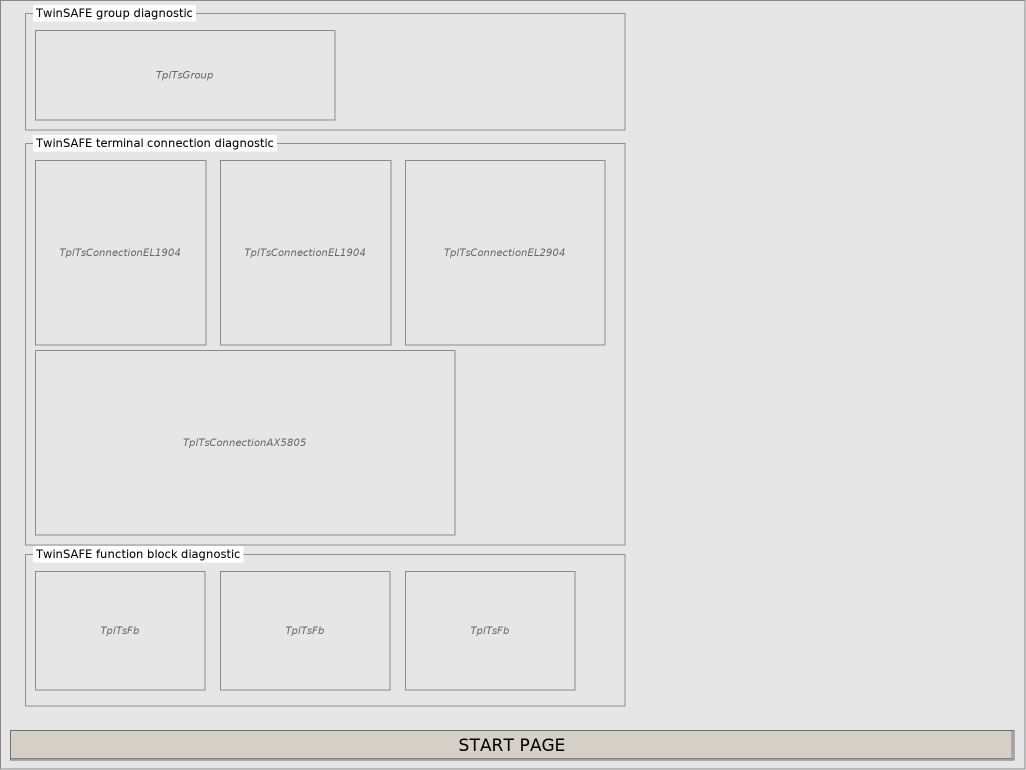
VISUALIZATION HmiTwinSAFEDiagnostic  // 1026x770
    Rectangle (0,0 1024x768)
    GroupBox (25,5 600x125), "TwinSAFE group diagnostic"
        Frame (10,25 300x90)
            shows TplTsGroup(stGroupDiag := TwinSAFE.fbSafeGroup1)
    GroupBox (25,135 600x410), "TwinSAFE terminal connection diagnostic"
        Frame (195,25 171x185)
            shows TplTsConnectionEL1904(stConnectionDiag := TwinSAFE.fbSafeConnectionEL1904_2_Group1)
        Frame (380,25 200x185)
            shows TplTsConnectionEL2904(stConnectionDiag := TwinSAFE.fbSafeConnectionEL2904_1_Group1)
        Frame (10,25 171x185)
            shows TplTsConnectionEL1904(stConnectionDiag := TwinSAFE.fbSafeConnectionEL1904_1_Group1)
        Frame (10,215 420x185)
            shows TplTsConnectionAX5805(stConnectionDiag := TwinSAFE.fbSafeConnectionAX5805_1_Group1)
    GroupBox (25,546 600x160), "TwinSAFE function block diagnostic"
        Frame (10,25 170x119)
            shows TplTsFb(stfbDiag := TwinSAFE.fbSafeFB_1_Group1)
        Frame (195,25 170x119)
            shows TplTsFb(stfbDiag := TwinSAFE.fbSafeFB_2_Group1)
        Frame (380,25 170x119)
            shows TplTsFb(stfbDiag := TwinSAFE.fbSafeFB_3_Group1)
    Button (10,730 1004x30), "START PAGE"
        OnMouseClick: change screen: HmiStartPage
END_VISUALIZATION

(* stored: Version 1.1.0.1, ProductVersion 3.1.4024.11
   Visu HmiTwinSAFEDiagnostic: Id {7cfcf2ba-eefd-4d4b-9e6a-65a1379ff497} *)
